{attribute 'qualified_only'}
VAR_GLOBAL
	ToStation: typeRemote;

END_VAR

(* stored: Version 1.1.0.1, ProductVersion 3.1.4024.12
   GVL Remote: Id {0cd9502d-d5ea-4a11-87aa-63e44e107acf} *)
